TYPE DUT_GetBatchHistoryDetail:
STRUCT  
	return_value	: DINT;
	BatchId			: STRING(50);
END_STRUCT
END_TYPE

(* stored: Version 1.1.0.1, ProductVersion 3.1.4024.15
   DUT DUT_GetBatchHistoryDetail: Id {0fb1d001-1602-405e-9b8c-a2e6890f3995} *)
